FUNCTION_BLOCK abstract FB_UniversalVFDModbus EXTENDS FB_ModbusSlaveRtu IMPLEMENTS I_UniversalVFD
VAR
	eVfdState	: E_Vfd_State;
	bInit	: BOOL;
	bBusy	: BOOL;
	bReset	: BOOL;
	bStop	: BOOL;
	bAbort : BOOL;
	bWarning : BOOL;// status
	bRunningForward	: BOOL;// in state running forward
	bRunningReverse	: BOOL; // in state running reverse
	bRanForward	: BOOL;
	bRanReverse	: BOOL;
	lrHzActual	: LREAL;
	lrDcVoltage		: LREAL;
	lrVacOutToMotor	: LREAL;
	lrCurrent	: LREAL;	
	lrPowerKw	: LREAL;	
	eVfdStatus	: E_VFD_Status;
	lrHzControl	: LREAL;// value in range(0.0-50.0Hz)
	iErrorID		: UDINT;

	lrSpeed : LREAL;
	lrTorque : LREAL;
	lrTotalKwh : LREAL;
	lrRatedPower : LREAL;
	bActive: BOOL;
	bOverLoad: BOOL;
	bStopLog: BOOL;
	bStopped: BOOL;
	
	VFD_CTRL_RESET_FAULT : WORD;
	VFD_CTRL_RUN_FORWARD :WORD;
	VFD_CTRL_RUN_REVERSE :WORD ;
	VFD_CTRL_STOP_FREE 	:WORD ;
	VFD_CTRL_STOP_SPEED_DOWN :WORD ;
	
	tonStopDelay: Ton;
	// time delay after status = stop
	tStopDelay: TIME := T#4S;
END_VAR
VAR CONSTANT
	// index
	iCTRL_WORD	: UINT := 1;
	iCTRL_FREQUENCY_WORD :UINT := 0;
	iSTATUS_WORD	: UINT := 0;
END_VAR

StateMachine();
CASE eVfdStatus OF
	VFD_STATUS_RUNNING_FORWARD :
		bRanForward := TRUE;
		bRanReverse := FALSE;
		bStopped := FALSE;
	VFD_STATUS_RUNNING_REVERSE:
		bRanForward := FALSE;
		bRanReverse := TRUE;
		bStopped := FALSE;
	VFD_STATUS_FAULT,VFD_STATUS_STOP:
		bRanForward := FALSE;
		bRanReverse := FALSE;
		bStopped := TRUE;
		
END_CASE
bError := eVfdStatus = VFD_STATUS_FAULT;
bActive := eVfdState >= VFD_IDLE;
SUPER^();
CASE eVfdState OF
	VFD_INITIALIZING..VFD_RESET_DONE, VFD_ABORTING:
		tonConfirmReallyError(
			IN := bError OR bModbusError,
			PT := timeConfirmReallyError,
			Q => bReallyError 
		);
END_CASE

{attribute 'monitoring' := 'variable'}
PROPERTY Active : REFERENCE TO  bool
GET
Active REF= bActive;
END_GET
END_PROPERTY

PROPERTY AcVoltageToMotor : Reference to lreal
GET
AcVoltageToMotor ref= lrVacOutToMotor;
END_GET
END_PROPERTY

{attribute 'monitoring' := 'variable'}
PROPERTY Busy : reference to bool
GET
Busy ref= bBusy;
END_GET
END_PROPERTY

METHOD Convert : BOOL
VAR_INPUT
	iRegionNo	:	INT;
	pReadData	:	POINTER TO word;
END_VAR
(*CASE iRegionNo OF
	0:
		// Status word
		Inverter_Ready		:=  pReadData[0].0;
		InverterReadyToRun	:=  pReadData[0].1;
		InverterRunning		:=  pReadData[0].2;
		InverterFaultActive :=  pReadData[0].3;
		OFF2_active			:= NOT pReadData[0].4;
		OFF3_active			:= NOT  pReadData[0].5;
		ON_inhibit_active 	 := pReadData[0].6;
		Inverter_warning_active := pReadData[0].7;
		Deviation_setpoint_OR_ActiveValue := NOT pReadData[0].8;
		PZD_control 		:= pReadData[0].9;
		Motor_current_Or_torque_limit  := NOT pReadData[0].11;
		Brake_open	 := pReadData[0].12;
		Motor_overload := NOT pReadData[0].13;
		Motor_RunRight	:= pReadData[0].14;
		Inverter_overload :=  NOT pReadData[0].15;
		
		IF InverterFaultActive THEN
			eStatus := VFD_STATUS_FAULT;
		ELSIF InverterFaultActive THEN
			eStatus := VFD_STATUS_WARNING;
		ELSIF InverterRunning THEN
			IF Motor_RunRight THEN
				eStatus := VFD_STATUS_RUNNING_FORWARD;
			ELSE
				eStatus := VFD_STATUS_RUNNING_REVERSE;
			END_IF
		ELSIF NOT InverterRunning THEN
			eStatus := VFD_STATUS_STOP;
		END_IF

		// Speed word
		lrHz_actual := WORD_TO_LREAL( pReadData[1])*50/16383;
		
	1:
		///  actual  Speed ( rpm) (unit A : Scale factor 1), Current ( A , 100, , Torque (Nm, 100)
	//, Actual Power (kw, 100), Total Kwh( 1), Dc bus Voltage(1), REFERENCE( hz, 100), RATED PWR( 100),OUTPUT VOLTS(1)
		lrSpeed := pReadData[0];
		lrCurrent := WORD_TO_LREAL(pReadData[1])/100;
		lrTorque := WORD_TO_LREAL(pReadData[2])/100;
		lrPower := WORD_TO_LREAL(pReadData[3])/100;
		lrTotalKwh := WORD_TO_LREAL(pReadData[4]);
		lrDc_Voltage := WORD_TO_LREAL(pReadData[5]);
		lrRatedPower := WORD_TO_LREAL(pReadData[7])/100;
		lrVAC_OutToMotor := WORD_TO_LREAL(pReadData[8]);
END_CASE
*)
END_METHOD

PROPERTY Current : reference to lreal
GET
Current ref= lrCurrent;
END_GET
END_PROPERTY

PROPERTY DcVoltage : Reference to lreal
GET
DcVoltage ref= lrDcVoltage;
END_GET
END_PROPERTY

{attribute 'monitoring' := 'variable'}
PROPERTY ErrorID : reference to UDINT
GET
ErrorID ref= iErrorID;
END_GET
END_PROPERTY

METHOD  FirstCycle 
VAR_INPUT
	sName : STRING;
	iUnitID : BYTE ; // modbus address of the device : 1- 255
END_VAR
THIS^.sName := sName;
THIS^.iUnitID := iUnitID;
(*(*HSW (speed setpoint), HIW (actual speed), STW (control word), ZSW (status word) refer to
control data. For more information, see parameters r2018 and P2019 in Chapter "Parameter
list (Page 147)*)
//ZSW  (status WORD), HIW (actual speed)
	arrAddress[0][0] := 109;
	arrAddress[0][1]	:= 2;

///  actual  Speed ( rpm) (unit A : Scale factor 1), Current ( A , 100, , Torque (Nm, 100)
	//, Actual Power (kw, 100), Total Kwh( 1), Dc bus Voltage(1), REFERENCE( hz, 100), RATED PWR( 100),OUTPUT VOLTS(1)
	arrAddress[1][0] := 24;
	arrAddress[1][1] := 10;

	
iNumAddRegion	:= 2;
/////write control  VFD
	
// Frequency

arrAddressWrite[0][0]	:= 100;
arrAddressWrite[0][1] 	:= 1;
arrAddressWrite[0][2]	:= LREAL_TO_WORD( FC_ScaleValue(	rangeRawMin := 0,
															rangeRawMax := 50,
															RangeScaleMin :=0,
															RangeScaleMax := 16384,
															ValueRaw := lrHz_Control) );
// Control word																	
arrAddressWrite[1][0]	:= 99;
arrAddressWrite[1][1] := 1;
arrAddressWrite[1][2]	:= 1150; //VFD_CTRL_STOP_SPEED_DOWN
iNumAddRegionWrite := 2;
*)
END_METHOD

PROPERTY HzActual : REFERENCE TO  LReal
GET
HzActual ref= lrHzActual;
END_GET
END_PROPERTY

PROPERTY HzControl : reference to LReal
GET
HzControl ref= lrHzControl;
END_GET
END_PROPERTY

{attribute 'monitoring' := 'variable'}
PROPERTY InHz : bool
GET
InHz :=  F_InRange( bound1 := lrHzControl +1,
					bound2 := lrHzControl -1,
					value := lrHzActual) ;
END_GET
END_PROPERTY

PROPERTY isRunForward : bool
GET
isRunForward := bRanForward;
END_GET
END_PROPERTY

{attribute 'monitoring' := 'variable'}
PROPERTY IsRunning : bool
GET
IsRunning := eVfdStatus = VFD_STATUS_RUNNING_FORWARD
			 OR  eVfdStatus = VFD_STATUS_RUNNING_REVERSE;
END_GET
END_PROPERTY

PROPERTY isRunReverse : bool
GET
isRunReverse := bRanReverse;
END_GET
END_PROPERTY

PROPERTY isStop : bool
GET
isStop := bStopped;
END_GET
END_PROPERTY

METHOD MR_Abort : BOOL
VAR_INPUT
END_VAR
IF eVfdState >= VFD_INITIALIZING THEN
	bAbort := TRUE;
	eVfdState := VFD_ABORTING;
	fbMachineLogger.MR_AddLogs(CONCAT(sName,' : abort requested'));
	bBusy := TRUE;
	
ELSIF eVfdState = VFD_UNINITIALIZED THEN
	bAbort 		:= FALSE;
	MR_Abort	:= TRUE;
	bBusy := FALSE;
	fbMachineLogger.MR_AddLogs(CONCAT(sName,' : abort done'));
	
END_IF
END_METHOD

METHOD MR_Init : bool
VAR_INPUT
END_VAR
IF eVFDState = VFD_UNINITIALIZED THEN
	bInit := TRUE;
	MR_Init := FALSE;
	eVfdState := VFD_INITIALIZING;
	fbMachineLogger.MR_AddLogs(CONCAT(sName,' : initialization requested'));
	bBusy := TRUE;
	
ELSIF eVFDState = VFD_READY_INITIALIZED THEN
	bInit := FALSE;
	MR_Init := TRUE;
	bBusy := FALSE;
	fbMachineLogger.MR_AddLogs(CONCAT(sName,' : initialization done'));
END_IF
END_METHOD

METHOD MR_Reset : BOOL
VAR_INPUT
END_VAR
IF eVfdState >= VFD_IDLE AND bError THEN
	bReset := TRUE;
	eVfdState := VFD_RESET;
	fbMachineLogger.MR_AddLogs(CONCAT(sName,' : reset requested'));			
	bBusy := TRUE;
	
ELSIF eVfdState = VFD_RESET_DONE THEN
	bError := FALSE;
	iErrorID := 0;
	bReset := FALSE;
	MR_Reset := TRUE;
	bBusy := FALSE;
	fbMachineLogger.MR_AddLogs(CONCAT(sName,' : reset done'));		
		
END_IF
END_METHOD

METHOD MR_RunForward : BOOL
VAR_INPUT
	hz : LREAL; 
END_VAR
IF eVfdState = VFD_IDLE  AND (NOT  F_InRange( 	bound1 := lrHzControl + 0.01,
												bound2 := lrHzControl - 0.01,
												value :=  hz)
								OR bRanReverse
								OR bStopped)
THEN
	lrHzControl := hz;
	bRunningForward := TRUE;
	MR_RunForward := FALSE;
	eVfdState := VFD_RUN_FORWARD;
	fbMachineLogger.MR_AddLogs( sLogMessage := FUN_MergeStrings4(  sName,' : run ',LREAL_TO_STRING( lrHzControl),' forward requested'));		
	bBusy := TRUE;
	
ELSIF eVfdState = VFD_RUN_FORWARD_DONE THEN
	bRunningForward := FALSE;
	MR_RunForward := TRUE;
	fbMachineLogger.MR_AddLogs(CONCAT(sName,' : run forward done'));	
	bBusy := FALSE;
END_IF
END_METHOD

METHOD MR_RunReverse : BOOL// must stop before call run reverse or forward
VAR_INPUT
	hz : LREAL; // >0 and < 50;
END_VAR
IF eVfdState = VFD_IDLE  AND (NOT  F_InRange( 	bound1 := lrHzControl + 0.01,
												bound2 := lrHzControl - 0.01,
												value :=  hz)
								OR bRanForward
								OR bStopped)
THEN
	lrHzControl := hz;
	bRunningReverse := TRUE;
	MR_RunReverse := FALSE;
	eVfdState := VFD_RUN_REVERSE;
	fbMachineLogger.MR_AddLogs( sLogMessage := FUN_MergeStrings4(  sName,' : run ',LREAL_TO_STRING( lrHzControl),' forward requested'));		
	bBusy := TRUE;
	
ELSIF eVfdState = VFD_RUN_REVERSE_DONE THEN
	bRunningReverse := FALSE;
	MR_RunReverse := TRUE;
	fbMachineLogger.MR_AddLogs(CONCAT(sName,' : run forward done'));
	bBusy := FALSE;
END_IF
END_METHOD

METHOD MR_Stop : BOOL
VAR_INPUT
END_VAR
IF eVfdState >= VFD_IDLE 
	AND eVfdState <> VFD_STOP_DONE
	AND NOT bStopped
THEN
	IF NOT bStopLog THEN 
		fbMachineLogger.MR_AddLogs(CONCAT(sName,' : stop requested'));
		bStopLog := TRUE;	
	END_IF
	
	bStop := TRUE;
	eVfdState := VFD_STOP;
	bBusy := TRUE;
	
ELSIF eVfdState = VFD_STOP_DONE THEN
	bStop 		:= FALSE;
	MR_Stop 	:= TRUE;
	bStopLog 	:= FALSE;
	fbMachineLogger.MR_AddLogs(CONCAT(sName,' : stop done'));	
	bBusy := FALSE;
END_IF
END_METHOD

METHOD PROTECTED MS_Aborting
lrHzControl := 0;
bInit := FALSE;
bRunningForward := FALSE;
bRunningReverse := FALSE;
bReset := FALSE;
bRanForward := FALSE;
bRanReverse := FALSE;
bOverLoad := FALSE;
bStop := FALSE;
bStopLog := FALSE;
bStopped := FALSE;
THIS^.tonStopDelay(IN :=FALSE);
eVfdState := VFD_UNINITIALIZED;
END_METHOD

METHOD PROTECTED MS_Idle
;
END_METHOD

METHOD  PROTECTED  MS_Initializing
// from Subclass call Super^.MS_Initializing
arrAddressWrite[iCTRL_WORD][2]	:= VFD_CTRL_RESET_FAULT;
IF eVfdStatus = VFD_STATUS_READY_TO_RUN THEN
	eVFDState := VFD_READY_INITIALIZED;
END_IF
END_METHOD

METHOD PROTECTED MS_ReadyInitialized
VAR_INPUT
END_VAR
IF NOT bInit THEN
	eVfdState := VFD_IDLE;
END_IF
END_METHOD

METHOD PROTECTED  MS_Reset
VAR_INPUT
END_VAR
arrAddressWrite[iCTRL_WORD][2]	:= VFD_CTRL_RESET_FAULT;
IF THIS^.evfdStatus <>  VFD_STATUS_NOT_RESPOND AND
	THIS^.evfdStatus <>  VFD_STATUS_FAULT THEN
	evfdState := VFD_RESET_DONE;
END_IF
END_METHOD

METHOD PROTECTED MS_ResetDone
VAR_INPUT
END_VAR
IF NOT bReset THEN
	evfdState := VFD_IDLE;
END_IF
END_METHOD

METHOD PROTECTED  MS_RunForward
VAR_INPUT
END_VAR
(*arrAddressWrite[iCtrlFrequencyWord][2] :=  LREAL_TO_WORD( 
											FC_ScaleValue(		rangeRawMin := 0,
																rangeRawMax := 50,
																RangeScaleMin := WORD_TO_LREAL( wHzWordValueMin),
																RangeScaleMax := WORD_TO_LREAL( wHzWordValueMax),
																ValueRaw := lrHzControl) 
														);*)
arrAddressWrite[iCTRL_WORD][2]	:= VFD_CTRL_RUN_FORWARD;
IF eVfdStatus = VFD_STATUS_RUNNING_FORWARD 
(*AND F_InRange( bound1 := lrHzControl + 1,
				bound2 := lrHzControl -1,
				value := lrHzActual)*)
THEN
	eVFDState := VFD_RUN_FORWARD_DONE;
END_IF
END_METHOD

METHOD PROTECTED MS_RunForwardDone
IF NOT bRunningForward THEN
	eVfdState := VFD_IDLE;
END_IF
END_METHOD

METHOD PROTECTED  MS_RunReverse
VAR_INPUT
END_VAR
(*arrAddressWrite[iCtrlFrequencyWord][2] :=  LREAL_TO_WORD( 
											FC_ScaleValue(		rangeRawMin := 0,
																rangeRawMax := 50,
																RangeScaleMin := WORD_TO_LREAL( wHzWordValueMin),
																RangeScaleMax := WORD_TO_LREAL( wHzWordValueMax),
																ValueRaw := lrHzControl) 
														);*)
arrAddressWrite[iCTRL_WORD][2]	:= VFD_CTRL_RUN_REVERSE;
IF eVfdStatus = VFD_STATUS_RUNNING_REVERSE 
(*AND F_InRange( bound1 := lrHzControl + 1,
				bound2 := lrHzControl -1,
				value := lrHzActual)*)
THEN
	eVFDState := VFD_RUN_REVERSE_DONE;
END_IF
END_METHOD

METHOD PROTECTED MS_RunReverseDone
VAR_INPUT
END_VAR
IF NOT bRunningReverse THEN
	eVfdState := VFD_IDLE;
END_IF
END_METHOD

METHOD protected  MS_Stop 
VAR_INPUT
END_VAR
arrAddressWrite[iCTRL_WORD][2]	:= VFD_CTRL_STOP_SPEED_DOWN;
(*tonStopDelay( in := eVfdStatus = VFD_STATUS_STOP,
				PT := tStopDelay);*)
IF eVfdStatus = VFD_STATUS_STOP THEN
 eVfdState := VFD_STOP_DONE;	
END_IF
(*IF tonStopDelay.Q THEN
	tonStopDelay(IN := FALSE);
	
END_IF*)
END_METHOD

METHOD protected Ms_StopDone
VAR_INPUT
END_VAR
IF NOT bStop THEN
	eVfdState := VFD_IDLE;
END_IF
END_METHOD

METHOD PROTECTED MS_Uninitialized
END_METHOD

{attribute 'monitoring' := 'variable'}
PROPERTY Overload : reference TO BOOL
GET
Overload REF= bOverLoad;
END_GET
END_PROPERTY

{attribute 'monitoring' := 'variable'}
PROPERTY PowerKw : REFERENCE TO LREAL
GET
PowerKw ref= lrPowerKw;
END_GET
END_PROPERTY

PROPERTY Speed : Reference to lreal
GET
Speed REF= lrSpeed;
END_GET
END_PROPERTY

{attribute 'monitoring' := 'variable'}
PROPERTY State : reference to E_Vfd_State
GET
State REF= eVfdState;
END_GET
END_PROPERTY

METHOD PROTECTED StateMachine
CASE eVfdState OF
	VFD_UNINITIALIZED :
		MS_Uninitialized();
		
	VFD_INITIALIZING	:
		MS_Initializing();
		
	VFD_READY_INITIALIZED :
		MS_ReadyInitialized();
		
	VFD_IDLE:
		MS_Idle();
	
	VFD_RUN_FORWARD	:
		MS_RunForward();
		
	VFD_RUN_FORWARD_DONE:
		MS_RunForwardDone();
	
	VFD_RUN_REVERSE	:
		MS_RunReverse();
	
	VFD_RUN_REVERSE_DONE:
		MS_RunReverseDone();
	
	VFD_STOP		:
		MS_Stop();
		
	VFD_STOP_DONE	:
		Ms_StopDone();
		
	VFD_RESET	:
		MS_Reset();
		
	VFD_RESET_DONE	:
		MS_ResetDone();
		
	VFD_ABORTING :
		MS_Aborting();
	
	
END_CASE
END_METHOD

{attribute 'monitoring' := 'variable'}
PROPERTY Status : reference to E_VFD_Status
GET
Status REF= eVfdStatus;
END_GET
END_PROPERTY

PROPERTY timeStopDelay : time
GET
timeStopDelay := THIS^.tStopDelay;
END_GET
SET
tStopDelay := timeStopDelay;
END_SET
END_PROPERTY

PROPERTY Torque : reference to lreal
GET
Torque ref= Torque;
END_GET
END_PROPERTY

PROPERTY TotalKwh : reference to lreal
GET
TotalKwh REF= TotalKwh;
END_GET
END_PROPERTY

// not all vfd modbus available this function 
PROPERTY Warning : reference to bool
GET
Warning  ref= bWarning;
END_GET
END_PROPERTY

END_FUNCTION_BLOCK

(* stored: Version 1.1.0.1, ProductVersion 3.1.4024.12
   POU FB_UniversalVFDModbus: Id {fd8d6acc-7bd2-4bb5-8c89-f74852cd1b9f}, SpecialFunc None
   Folder MR: Id {f3a3e522-a81c-41cc-b27b-dd5d55174206}
   Folder MS: Id {3c98f81a-bb00-4ab4-8c00-b47b98f5a50e}
   Folder Pro: Id {7c18a100-0569-4c54-a015-9f1f8eff674a}
   Property Active: Id {248f35d9-0534-4079-b983-4dfb71e4f83d}
   Get Get: Id {2e5b10b5-ecb5-4334-9ad9-62ac8d555930}
   Property AcVoltageToMotor: Id {e040051a-2a43-46a0-8a44-7b0b368e71d6}
   Get Get: Id {a75c5611-9da0-4952-a9d8-2818606333c5}
   Property Busy: Id {bfb2da44-65c7-4e0a-8206-1b28790c7fa7}
   Get Get: Id {3fa3786e-bf57-47d1-8f99-4ea0fcc21d83}
   Method Convert: Id {8638a3f3-4263-4048-a86b-3983221cb27f}
   Property Current: Id {df2898d1-d53c-4e49-bebf-d9596acf7350}
   Get Get: Id {7840d247-f7a3-4d31-a41e-327be16de82f}
   Property DcVoltage: Id {4b0563e7-60d5-45c0-80ed-6cb8218ead30}
   Get Get: Id {4163d4e2-2c56-4214-9300-5989979b2849}
   Property ErrorID: Id {96a1ef08-7d27-43d5-95f8-384722c0cd2f}
   Get Get: Id {7a2d77ea-644e-4d09-9c4f-06ff24296237}
   Method FirstCycle: Id {d0749a6c-4309-4783-9ca6-eadbfcd7d7b7}
   Property HzActual: Id {085f7d57-1175-4177-92fc-d0932167f162}
   Get Get: Id {17cdfd9c-9186-4c43-9e6d-8ffe2a39adb1}
   Property HzControl: Id {92a91086-914b-4bad-84ee-8590914bbbe8}
   Get Get: Id {80939dba-77b0-4c70-b414-7c310cf240e2}
   Property InHz: Id {bd6a5744-d2d1-4bbb-9451-991472a8a079}
   Get Get: Id {c50da6e4-adab-4e42-9c1a-3d616d5562e0}
   Property isRunForward: Id {530022fc-b0a8-4067-9ca0-5f623dadd3d2}
   Get Get: Id {8eca8758-3a5d-49bd-a784-190aa5ead541}
   Property IsRunning: Id {b530bfa5-e84e-408c-aaaa-7e1f96e8a90a}
   Get Get: Id {2db6c004-a6da-4278-8c46-b645d6af7143}
   Property isRunReverse: Id {a1b5a0e9-3535-416a-a324-64b2ed62421d}
   Get Get: Id {cf60e44f-322e-47d7-bc00-e9e3374faefb}
   Property isStop: Id {b2dcf4c1-7e4c-4950-aa01-317f8dff1fe0}
   Get Get: Id {8450012d-8bd8-4bb0-9ce2-31b14828a8b6}
   Method MR_Abort: Id {0652cd1f-8358-436c-b6d6-cd2b3c63779c}
   Method MR_Init: Id {10f4ed1f-54f3-4350-ae84-73832517b609}
   Method MR_Reset: Id {bf1dc21b-2f7f-4436-a1dc-6876cbe34721}
   Method MR_RunForward: Id {f2f3dd06-bdd8-4d87-b04a-6208e4158e93}
   Method MR_RunReverse: Id {60b3c7e3-bfe7-4f56-a3de-0900b804ca81}
   Method MR_Stop: Id {5154dd24-3d5c-4d9f-bc6e-ecd7665c5f2a}
   Method MS_Aborting: Id {ad704b6c-09e0-4c8a-89dd-99c32b7d53a4}
   Method MS_Idle: Id {39ad5f92-ecc8-4350-8dcc-ea7c447fca61}
   Method MS_Initializing: Id {824ac014-d11e-437b-82ec-de23cf38f6ee}
   Method MS_ReadyInitialized: Id {37e63d86-802f-406d-b8f9-5ae975bdc272}
   Method MS_Reset: Id {f0d93329-f152-4fd2-8c7f-871b868d0feb}
   Method MS_ResetDone: Id {80e652ac-4a03-414c-a1ef-06420ec2c202}
   Method MS_RunForward: Id {82195713-76f3-44d4-af66-4e860180a0ce}
   Method MS_RunForwardDone: Id {4d3ed909-9988-4d27-b6a5-98918b4e0b34}
   Method MS_RunReverse: Id {22900e6c-e0c2-4cba-a7e4-7cb557ba4e9e}
   Method MS_RunReverseDone: Id {cf1e0f42-763e-4c75-ac70-f2d87ce26a28}
   Method MS_Stop: Id {65edc64e-45a2-4831-b125-cccd979efc34}
   Method Ms_StopDone: Id {0b119057-c48d-4681-b54d-50db7368ad87}
   Method MS_Uninitialized: Id {e57b3e42-d437-4da7-a50f-5afe089940cf}
   Property Overload: Id {5957236b-6615-4544-ba72-3c42899ddd6f}
   Get Get: Id {57c5f420-3551-4e5b-b71e-062edf3b530b}
   Property PowerKw: Id {48775f63-c7bf-4af7-8ac9-724f8f086574}
   Get Get: Id {df981b4e-1d41-4766-9c53-e333cd121628}
   Property Speed: Id {05b0b761-4d95-4629-aa5a-3dcdbc2dec00}
   Get Get: Id {e0273508-a395-4e45-8a9f-24350d25a6df}
   Property State: Id {eb02e7a2-65a3-4091-85a2-7853e4e76990}
   Get Get: Id {90203748-2e2d-4061-9cc9-8ff81bd63590}
   Method StateMachine: Id {a28b4839-7dea-4f43-a0dd-a64c5ad12c77}
   Property Status: Id {087bc722-873f-43f4-a3f0-ed4a230ad30f}
   Get Get: Id {6608a8ef-53ca-4b87-8606-c98444f8029e}
   Property timeStopDelay: Id {23956b3e-67a2-4d6d-800c-eee10a2f627e}
   Get Get: Id {4fd094a7-1d01-49a8-8f40-8267c8a3a85e}
   Set Set: Id {b6fa5949-2626-42d2-9c03-df63e61791c3}
   Property Torque: Id {3a714a99-fc23-4bf9-819f-f6995e3d8134}
   Get Get: Id {eb049a2d-804b-453d-9dcd-143614074192}
   Property TotalKwh: Id {df528c9e-51e4-4219-9b94-b69576dbef37}
   Get Get: Id {c57beb9d-1ecd-4ea2-96fa-6da7ee11f4a6}
   Property Warning: Id {b540e38b-08da-4ae3-8220-2847dbf23316}
   Get Get: Id {e83b75d1-a5fc-40fe-bc08-b5d167853f32} *)
